Universal Robots PolyScope program: external_control.urp

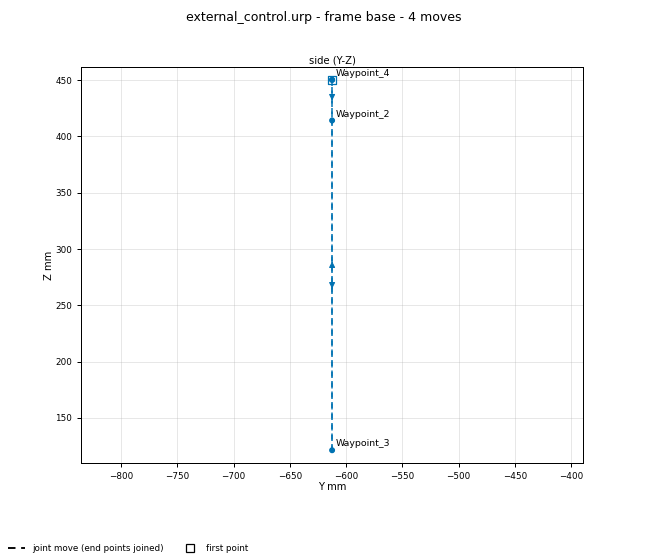
[picture p0: tool path of external_control.urp in frame base, 4 of 5 moves have a stored position in this frame; points joined in program order, loops and branches not executed]
Program external_control (installation=default directory=/home/mahp/ursim-5.9.1.1031110/programs createdIn=5.9.1.1031110 lastSavedIn=5.9.1.1031110 robotSerialNumber=20195599999)
Calibrated DH parameters: a=[0, -0.425, -0.3922, 0, 0, 0]; d=[0.1625, 0, 0, 0.1333, 0.0997, 0.0996]; alpha=[1.570796, 0, 0, 1.570796, -1.570796, 0]; deltaTheta=[0, 0, 0, 0, 0, 0]
Robot Program (runOnlyOnce=false)
  var_1 := get_actual_tcp_pose()
  MoveJ speed 60 deg/s, acceleration 80 deg/s^2 (useActiveTCP=true) feature=Base
    Waypoint Waypoint (Variable): variable=var_1
    Waypoint Waypoint_4: TCP in base x=-210.755 y=-612.435 z=450.305 mm, rx=2.8927 ry=1.0832 rz=0.0329 rad; joints [58.642, -70.835, 73.139, 266.797, -86.877, 107.611] deg
  URCap External Control (External Control, FZI Research Center for Information Technology)
  MoveJ speed 60 deg/s, acceleration 80 deg/s^2 (useActiveTCP=true) feature=Base
    Waypoint Waypoint_2: TCP in base x=-210.755 y=-612.435 z=414.205 mm, rx=2.8927 ry=1.0832 rz=0.0329 rad; joints [58.642, -70.408, 77.853, 261.656, -86.877, 107.611] deg
    Waypoint Waypoint_3: TCP in base x=-210.755 y=-612.435 z=121.263 mm, rx=2.8927 ry=1.0832 rz=0.0329 rad; joints [58.642, -52.633, 98.426, 223.308, -86.877, 107.611] deg
    Waypoint Waypoint_4: TCP in base x=-210.755 y=-612.435 z=450.305 mm, rx=2.8927 ry=1.0832 rz=0.0329 rad; joints [58.642, -70.835, 73.139, 266.797, -86.877, 107.611] deg
